SUBAPPLICATION QueryServiceOpcUaSubFull (* Query services using OPC UA with all service's fields to be defined *)
  (* Standard: 61499-2; Description: Copyright (c) 2019 fortiss GmbH This program and the accompanying materials are made available under the terms of the Eclipse Public License 2.0 which is available at https://www.eclipse.org/legal/epl-2.0/ SPDX-License-Identifier: EPL-2.0 *)
  (* Version 1.0, 2019-09-17, Jose Cabral, fortiss GmbH *)
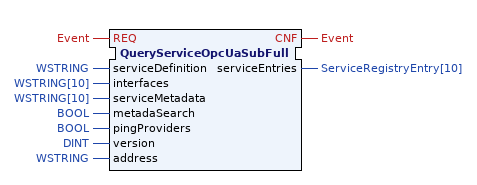
  EVENT_INPUT
    REQ; (* Query for services *)
  END_EVENT
  EVENT_OUTPUT
    CNF; (* Query finished *)
  END_EVENT
  VAR_INPUT
    serviceDefinition : WSTRING; (* Interfaces implemented by the service *)
    interfaces : ARRAY [0..9] OF WSTRING; (* Interfaces implemented by the service *)
    serviceMetadata : ARRAY [0..9] OF WSTRING; (* Metadata of the service in key=value format *)
    metadaSearch : BOOL; (* True, if service metadata shall be taken into account during query *)
    pingProviders : BOOL; (* True, if the selected (query fitting) Application Systems shall be pinged to see if they’re alive *)
    version : DINT; (* The minimum version of the Service we are looking for *)
    address : WSTRING; (* Address of the Service Registry *)
  END_VAR
  VAR_OUTPUT
    serviceEntries : ARRAY [0..9] OF ServiceRegistryEntry;
  END_VAR
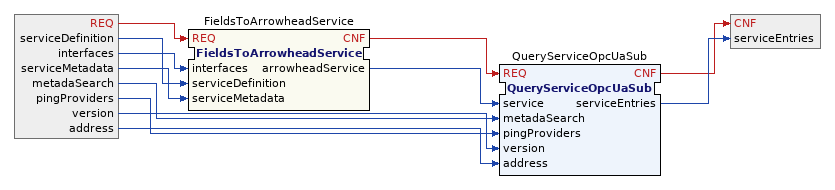
  FBS
    FieldsToArrowheadService : FieldsToArrowheadService;
  END_FBS
  SUBAPPS
    QueryServiceOpcUaSub : QueryServiceOpcUaSub;
  END_SUBAPPS
  EVENT_CONNECTIONS
    REQ TO FieldsToArrowheadService.REQ;
    FieldsToArrowheadService.CNF TO QueryServiceOpcUaSub.REQ;
    QueryServiceOpcUaSub.CNF TO CNF;
  END_CONNECTIONS
  DATA_CONNECTIONS
    interfaces TO FieldsToArrowheadService.interfaces;
    serviceDefinition TO FieldsToArrowheadService.serviceDefinition;
    serviceMetadata TO FieldsToArrowheadService.serviceMetadata;
    FieldsToArrowheadService.arrowheadService TO QueryServiceOpcUaSub.service;
    metadaSearch TO QueryServiceOpcUaSub.metadaSearch;
    pingProviders TO QueryServiceOpcUaSub.pingProviders;
    version TO QueryServiceOpcUaSub.version;
    address TO QueryServiceOpcUaSub.address;
    QueryServiceOpcUaSub.serviceEntries TO serviceEntries;
  END_CONNECTIONS
END_SUBAPPLICATION
